// TIA Portal project "FactoryIO_Template_S7-1500_V15" (V15)

(* hardware
DEVICE "S71500/ET200MP-Station_1"  S7-1500 station
   slot 0: "Profilschiene_0"  6ES7 590-1***0-0AA0
   slot 1: "PLC_1"  CPU 1511-1 PN  6ES7 511-1AK00-0AB0  V1.8
   slot 2: "AI 8xU/I/RTD/TC ST_1"  AI 8xU/I/RTD/TC ST  6ES7 531-7KF00-0AB0  V2.0
   slot 3: "AI 8xU/I/RTD/TC ST_2"  AI 8xU/I/RTD/TC ST  6ES7 531-7KF00-0AB0  V2.0
   slot 4: "AI 8xU/I/RTD/TC ST_3"  AI 8xU/I/RTD/TC ST  6ES7 531-7KF00-0AB0  V2.0
   slot 5: "AI 8xU/I/RTD/TC ST_4"  AI 8xU/I/RTD/TC ST  6ES7 531-7KF00-0AB0  V2.0
   slot 6: "DI 16x24VDC BA_1"  DI 16x24VDC BA  6ES7 521-1BH10-0AA0  V1.0
*)

// ===== PLC "PLC_1"  CPU 1511-1 PN =====

VAR_GLOBAL   // PLC tag table "Standard-Variablentabelle"
   "counter green" AT %QD31 : UDInt;
END_VAR

VAR_GLOBAL   // PLC tag table "Input tag table"
   "start" AT %I0.0 : Bool;
   "stop" AT %I0.1 : Bool;
   "reset" AT %I0.2 : Bool;
   "emergency" AT %I0.3 : Bool;
   "right 1 limit" AT %I0.4 : Bool;
   "right 1 clamped" AT %I0.5 : Bool;
   "right 2 limit" AT %I0.6 : Bool;
   "right 2 clamped" AT %I0.7 : Bool;
   "mc1 opened" AT %I1.0 : Bool;
   "mc1 busy" AT %I1.1 : Bool;
   "mc1 error" AT %I1.2 : Bool;
   "mc2 opened" AT %I1.3 : Bool;
   "mc2 busy" AT %I1.4 : Bool;
   "mc2 error" AT %I1.5 : Bool;
   "mc3 opened" AT %I1.6 : Bool;
   "mc3 busy" AT %I1.7 : Bool;
   "mc3 error" AT %I2.0 : Bool;
   "mc5 opened" AT %I2.1 : Bool;
   "mc5 busy" AT %I2.2 : Bool;
   "mc5 error" AT %I2.3 : Bool;
   "pusher 3 front limit" AT %I2.4 : Bool;
   "pusher 1 front limit" AT %I2.5 : Bool;
   "pusher 4 front limit" AT %I2.6 : Bool;
   "pusher 2 front limit" AT %I2.7 : Bool;
   "right 3 limit" AT %I3.0 : Bool;
   "right 3 clamped" AT %I3.1 : Bool;
   "right 5 limit" AT %I3.2 : Bool;
   "right 5 clamped" AT %I3.3 : Bool;
   "axis 1 detected" AT %I3.4 : Bool;
   "axis 1 moving z" AT %I3.5 : Bool;
   "axis 1 moving x" AT %I3.6 : Bool;
   "axis 2 detected" AT %I3.7 : Bool;
   "axis 2 moving z" AT %I4.0 : Bool;
   "axis 2 moving x" AT %I4.1 : Bool;
   "vision sensor 1" AT %I4.2 : Bool;
   "vision sensor 2" AT %I4.3 : Bool;
   "vision sensor 3" AT %I4.4 : Bool;
   "vision sensor 4" AT %I4.5 : Bool;
   "diffuser sensor 1" AT %I4.6 : Bool;
   "diffuser sensor 2" AT %I4.7 : Bool;
   "diffuser sensor 3" AT %I5.0 : Bool;
   "diffuser sensor 4" AT %I5.1 : Bool;
   "diffuser sensor 5" AT %I5.2 : Bool;
   "diffuser sensor 6" AT %I5.3 : Bool;
END_VAR

VAR_GLOBAL   // PLC tag table "Memory tag table"
   "start memory" AT %M0.0 : Bool;
   "stop memory" AT %M0.1 : Bool;
   "Tag_1" AT %M0.2 : Bool;
   "Tag_2" AT %M0.3 : Bool;
   "Tag_3" AT %M0.4 : Bool;
   "Tag_4" AT %M0.5 : Bool;
   "Tag_5" AT %M0.6 : Bool;
   "Tag_6" AT %M0.7 : Bool;
   "Lid alined" AT %M1.0 : Bool;
   "Tag_7" AT %M1.1 : Bool;
   "Tag_8" AT %M1.2 : Bool;
   "base alined" AT %M1.3 : Bool;
   "Tag_9" AT %M1.4 : Bool;
   "MOVE Z BIT" AT %M1.5 : Bool;
   "Tag_10" AT %M1.6 : Bool;
   "Tag_11" AT %M1.7 : Bool;
   "Tag_12" AT %M2.0 : Bool;
   "Tag_13" AT %M2.1 : Bool;
   "Tag_14" AT %M2.2 : Bool;
   "MOVE Z BIT 2" AT %M2.3 : Bool;
   "Tag_15" AT %M2.4 : Bool;
   "TEMPORARY" AT %M2.5 : Bool;
   "Tag_16" AT %M2.6 : Bool;
   "TEMPORARY 2" AT %M2.7 : Bool;
   "Tag_17" AT %M3.0 : Bool;
   "Tag_1(1)" AT %M3.1 : Bool;
   "Tag_2(1)" AT %M3.2 : Bool;
   "Tag_3(1)" AT %M3.3 : Bool;
   "Tag_4(1)" AT %M3.4 : Bool;
   "Tag_5(1)" AT %M3.5 : Bool;
   "Tag_6(1)" AT %M3.6 : Bool;
   "Lid alined(1)" AT %M3.7 : Bool;
   "Tag_7(1)" AT %M4.0 : Bool;
   "Tag_8(1)" AT %M4.1 : Bool;
   "base alined(1)" AT %M4.2 : Bool;
   "Tag_9(1)" AT %M4.3 : Bool;
   "MOVE Z BIT(1)" AT %M4.4 : Bool;
   "Tag_10(1)" AT %M4.5 : Bool;
   "Tag_11(1)" AT %M4.6 : Bool;
   "Tag_12(1)" AT %M4.7 : Bool;
   "Tag_13(1)" AT %M5.0 : Bool;
   "Tag_14(1)" AT %M5.1 : Bool;
   "MOVE Z BIT 2(1)" AT %M5.2 : Bool;
   "Tag_15(1)" AT %M5.3 : Bool;
   "TEMPORARY(1)" AT %M5.4 : Bool;
   "Tag_16(1)" AT %M5.5 : Bool;
   "TEMPORARY 2(1)" AT %M5.6 : Bool;
   "Tag_17(1)" AT %M5.7 : Bool;
   "tag 18" AT %M6.0 : Bool;
END_VAR

VAR_GLOBAL   // PLC tag table "Output tag table"
   "belt conveyor (2m)1" AT %Q0.0 : Bool;
   "belt conveyor (2m)2" AT %Q0.1 : Bool;
   "belt conveyor (2m)3" AT %Q0.2 : Bool;
   "belt conveyor (2m)5" AT %Q0.3 : Bool;
   "belt conveyor (2m)7" AT %Q0.4 : Bool;
   "belt conveyor (2m)9" AT %Q0.5 : Bool;
   "belt conveyor (2m)14" AT %Q0.6 : Bool;
   "belt conveyor (4m)2" AT %Q1.0 : Bool;
   "belt conveyor (4m)4" AT %Q1.1 : Bool;
   "belt conveyor (6m)1" AT %Q1.2 : Bool;
   "emitter 2" AT %Q1.3 : Bool;
   "emitter 3" AT %Q1.4 : Bool;
   "emitter 4" AT %Q1.5 : Bool;
   "emitter 6" AT %Q1.6 : Bool;
   "factory pause" AT %Q1.7 : Bool;
   "factory reset" AT %Q2.0 : Bool;
   "right 1 clamp" AT %Q2.1 : Bool;
   "right 1 raise" AT %Q2.2 : Bool;
   "right 2 clamp" AT %Q2.3 : Bool;
   "right 2 raise" AT %Q2.4 : Bool;
   "mc1 start" AT %Q2.5 : Bool;
   "mc1 stop" AT %Q2.6 : Bool;
   "mc1 reset" AT %Q2.7 : Bool;
   "mc1 producing leds" AT %Q3.0 : Bool;
   "mc2 start" AT %Q3.1 : Bool;
   "mc2 stop" AT %Q3.2 : Bool;
   "mc2 reset" AT %Q3.3 : Bool;
   "mc2 producing leds" AT %Q3.4 : Bool;
   "mc3 start" AT %Q3.5 : Bool;
   "mc3 stop" AT %Q3.6 : Bool;
   "mc3 reset" AT %Q3.7 : Bool;
   "mc3 producing leds" AT %Q4.0 : Bool;
   "mc5 start" AT %Q4.1 : Bool;
   "mc5 stop" AT %Q4.2 : Bool;
   "mc5 reset" AT %Q4.3 : Bool;
   "mc5 producing leds" AT %Q4.4 : Bool;
   "pusher 1" AT %Q4.5 : Bool;
   "pusher 2" AT %Q4.6 : Bool;
   "remover 1" AT %Q4.7 : Bool;
   "remover 2" AT %Q5.0 : Bool;
   "reset light" AT %Q5.1 : Bool;
   "start light" AT %Q5.2 : Bool;
   "stop light" AT %Q5.3 : Bool;
   "right 3 clamp" AT %Q5.4 : Bool;
   "right 3 raise" AT %Q5.5 : Bool;
   "right 5 clamp" AT %Q5.6 : Bool;
   "right 5 raise" AT %Q5.7 : Bool;
   "axis 1 x" AT %Q6.0 : Bool;
   "axis 1 z" AT %Q6.1 : Bool;
   "axis 1 grab" AT %Q6.2 : Bool;
   "axis 2 x" AT %Q6.3 : Bool;
   "axis 2 z" AT %Q6.4 : Bool;
   "axis 2 grab" AT %Q6.5 : Bool;
   "belt conveyor (4m)1" AT %Q6.6 : Bool;
   "belt conveyor (6m)2" AT %Q6.7 : Bool;
   "belt conveyor (6m)3" AT %Q7.0 : Bool;
   "belt conveyor (6m)4" AT %Q7.1 : Bool;
   "belt conveyor (6m)5" AT %Q7.2 : Bool;
   "belt conveyor (6m)6" AT %Q7.3 : Bool;
   "pusher 3" AT %Q7.4 : Bool;
   "pusher 4" AT %Q7.5 : Bool;
   "counter blue" AT %QD8 : UDInt;
   "counter 2" AT %QD12 : UDInt;
END_VAR

// folder: System blocks/Program resources

DATA_BLOCK "IEC_Timer_0_DB"   // DB1
{ S7_Optimized_Access := 'TRUE' }
AUTHOR : Simatic
FAMILY : IEC
NAME : IEC_TMR
VERSION : 1.0
// stored: InstanceOfName IEC_TIMER
"IEC_TIMER"
BEGIN
END_DATA_BLOCK

DATA_BLOCK "IEC_Timer_0_DB_1"   // DB2
{ S7_Optimized_Access := 'TRUE' }
AUTHOR : Simatic
FAMILY : IEC
NAME : IEC_TMR
VERSION : 1.0
// stored: InstanceOfName IEC_TIMER
"IEC_TIMER"
BEGIN
END_DATA_BLOCK

DATA_BLOCK "IEC_Timer_0_DB_2"   // DB3
{ S7_Optimized_Access := 'TRUE' }
AUTHOR : Simatic
FAMILY : IEC
NAME : IEC_TMR
VERSION : 1.0
// stored: InstanceOfName IEC_TIMER
"IEC_TIMER"
BEGIN
END_DATA_BLOCK

DATA_BLOCK "IEC_Timer_0_DB_3"   // DB4
{ S7_Optimized_Access := 'TRUE' }
AUTHOR : Simatic
FAMILY : IEC
NAME : IEC_TMR
VERSION : 1.0
// stored: InstanceOfName IEC_TIMER
"IEC_TIMER"
BEGIN
END_DATA_BLOCK

DATA_BLOCK "IEC_Timer_0_DB_4"   // DB5
{ S7_Optimized_Access := 'TRUE' }
AUTHOR : Simatic
FAMILY : IEC
NAME : IEC_TMR
VERSION : 1.0
// stored: InstanceOfName IEC_TIMER
"IEC_TIMER"
BEGIN
END_DATA_BLOCK

DATA_BLOCK "IEC_Timer_0_DB_6"   // DB6
{ S7_Optimized_Access := 'TRUE' }
AUTHOR : Simatic
FAMILY : IEC
NAME : IEC_TMR
VERSION : 1.0
// stored: InstanceOfName IEC_TIMER
"IEC_TIMER"
BEGIN
END_DATA_BLOCK

// folder: (top level)

FUNCTION "blue belt conveyor" : Void   // FC1, LAD
{ S7_Optimized_Access := 'TRUE' }
VERSION : 0.1
   VAR_TEMP   // added for the SCL form of the ladder/FBD networks
      _w1 : Bool;
   END_VAR
BEGIN

REGION Network 1
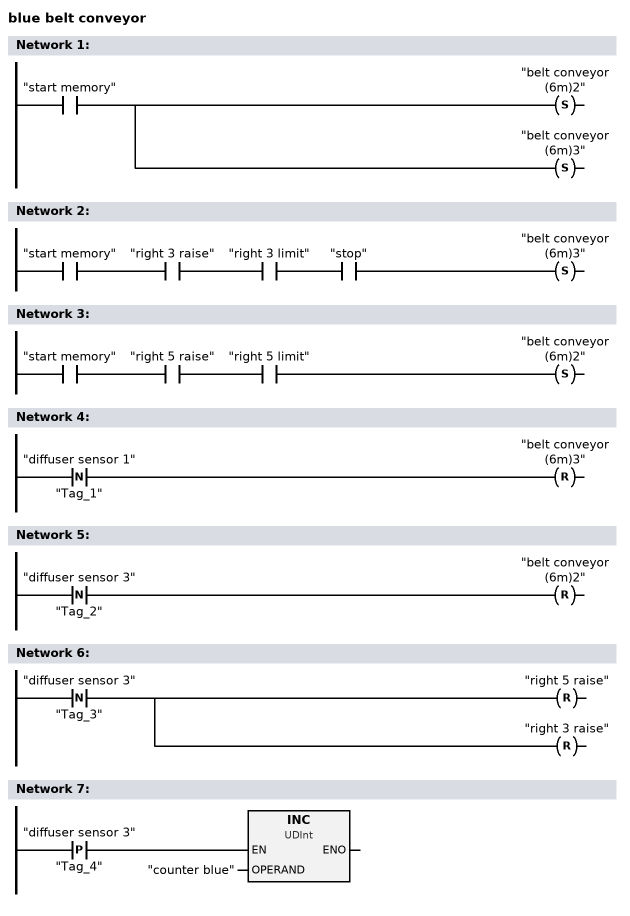
   RUNG wire#powerrail
      Contact( "start memory" )
      wire#w1
      S_Coil( "belt conveyor (6m)2" )
   END_RUNG
   RUNG wire#w1
      S_Coil( "belt conveyor (6m)3" )
   END_RUNG
   // the same network as SCL:
   IF "start memory" THEN
       "belt conveyor (6m)2" := TRUE;
       "belt conveyor (6m)3" := TRUE;
   END_IF;
END_REGION

REGION Network 2
   RUNG wire#powerrail
      Contact( "start memory" )
      Contact( "right 3 raise" )
      Contact( "right 3 limit" )
      Contact( "stop" )
      S_Coil( "belt conveyor (6m)3" )
   END_RUNG
   // the same network as SCL:
   IF "start memory" AND "right 3 raise" AND "right 3 limit" AND "stop" THEN
       "belt conveyor (6m)3" := TRUE;
   END_IF;
END_REGION

REGION Network 3
   RUNG wire#powerrail
      Contact( "start memory" )
      Contact( "right 5 raise" )
      Contact( "right 5 limit" )
      S_Coil( "belt conveyor (6m)2" )
   END_RUNG
   // the same network as SCL:
   IF "start memory" AND "right 5 raise" AND "right 5 limit" THEN "belt conveyor (6m)2" := TRUE; END_IF;
END_REGION

REGION Network 4
   RUNG wire#powerrail
      N_Contact(operand := "diffuser sensor 1", bit := "Tag_1")
      R_Coil( "belt conveyor (6m)3" )
   END_RUNG
   // the same network as SCL:
   #_w1 := NOT "diffuser sensor 1" AND "Tag_1";   // falling edge of "diffuser sensor 1"
   "Tag_1" := "diffuser sensor 1";
   IF #_w1 THEN "belt conveyor (6m)3" := FALSE; END_IF;
END_REGION

REGION Network 5
   RUNG wire#powerrail
      N_Contact(operand := "diffuser sensor 3", bit := "Tag_2")
      R_Coil( "belt conveyor (6m)2" )
   END_RUNG
   // the same network as SCL:
   #_w1 := NOT "diffuser sensor 3" AND "Tag_2";   // falling edge of "diffuser sensor 3"
   "Tag_2" := "diffuser sensor 3";
   IF #_w1 THEN "belt conveyor (6m)2" := FALSE; END_IF;
END_REGION

REGION Network 6
   RUNG wire#powerrail
      N_Contact(operand := "diffuser sensor 3", bit := "Tag_3")
      wire#w1
      R_Coil( "right 5 raise" )
   END_RUNG
   RUNG wire#w1
      R_Coil( "right 3 raise" )
   END_RUNG
   // the same network as SCL:
   #_w1 := NOT "diffuser sensor 3" AND "Tag_3";   // falling edge of "diffuser sensor 3"
   "Tag_3" := "diffuser sensor 3";
   IF #_w1 THEN
       "right 5 raise" := FALSE;
       "right 3 raise" := FALSE;
   END_IF;
END_REGION

REGION Network 7
   RUNG wire#powerrail
      P_Contact(operand := "diffuser sensor 3", bit := "Tag_4")
      { S7_Templates := "DestType := UDInt" } Inc( "counter blue" )
   END_RUNG
   // the same network as SCL:
   #_w1 := "diffuser sensor 3" AND NOT "Tag_4";   // rising edge of "diffuser sensor 3"
   "Tag_4" := "diffuser sensor 3";
   IF #_w1 THEN "counter blue" := "counter blue" + 1; END_IF;
END_REGION
END_FUNCTION

FUNCTION "blue Clamp" : Void   // FC2, LAD
{ S7_Optimized_Access := 'TRUE' }
VERSION : 0.1
   VAR_TEMP   // added for the SCL form of the ladder/FBD networks
      _w1 : Bool;
   END_VAR
BEGIN

REGION Network 1
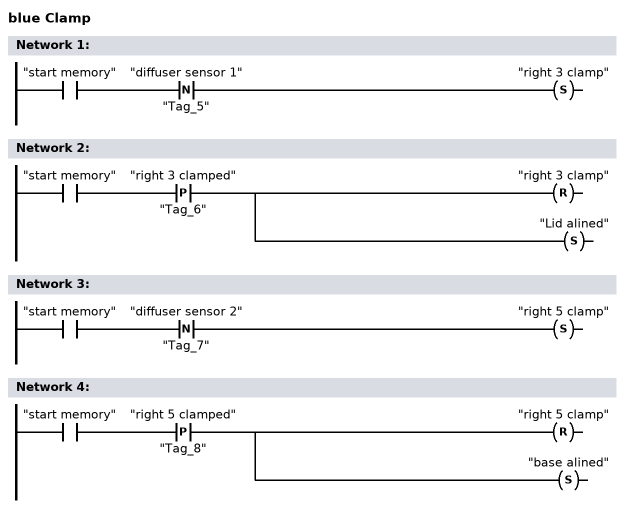
   RUNG wire#powerrail
      Contact( "start memory" )
      N_Contact(operand := "diffuser sensor 1", bit := "Tag_5")
      S_Coil( "right 3 clamp" )
   END_RUNG
   // the same network as SCL:
   #_w1 := "start memory" AND NOT "diffuser sensor 1" AND "Tag_5";   // falling edge of "diffuser sensor 1"
   "Tag_5" := "diffuser sensor 1";
   IF #_w1 THEN "right 3 clamp" := TRUE; END_IF;
END_REGION

REGION Network 2
   RUNG wire#powerrail
      Contact( "start memory" )
      P_Contact(operand := "right 3 clamped", bit := "Tag_6")
      wire#w1
      R_Coil( "right 3 clamp" )
   END_RUNG
   RUNG wire#w1
      S_Coil( "Lid alined" )
   END_RUNG
   // the same network as SCL:
   #_w1 := "start memory" AND "right 3 clamped" AND NOT "Tag_6";   // rising edge of "right 3 clamped"
   "Tag_6" := "right 3 clamped";
   IF #_w1 THEN
       "right 3 clamp" := FALSE;
       "Lid alined" := TRUE;
   END_IF;
END_REGION

REGION Network 3
   RUNG wire#powerrail
      Contact( "start memory" )
      N_Contact(operand := "diffuser sensor 2", bit := "Tag_7")
      S_Coil( "right 5 clamp" )
   END_RUNG
   // the same network as SCL:
   #_w1 := "start memory" AND NOT "diffuser sensor 2" AND "Tag_7";   // falling edge of "diffuser sensor 2"
   "Tag_7" := "diffuser sensor 2";
   IF #_w1 THEN "right 5 clamp" := TRUE; END_IF;
END_REGION

REGION Network 4
   RUNG wire#powerrail
      Contact( "start memory" )
      P_Contact(operand := "right 5 clamped", bit := "Tag_8")
      wire#w1
      R_Coil( "right 5 clamp" )
   END_RUNG
   RUNG wire#w1
      S_Coil( "base alined" )
   END_RUNG
   // the same network as SCL:
   #_w1 := "start memory" AND "right 5 clamped" AND NOT "Tag_8";   // rising edge of "right 5 clamped"
   "Tag_8" := "right 5 clamped";
   IF #_w1 THEN
       "right 5 clamp" := FALSE;
       "base alined" := TRUE;
   END_IF;
END_REGION
END_FUNCTION

FUNCTION "blue pICK & pLACE" : Void   // FC3, LAD
{ S7_Optimized_Access := 'TRUE' }
VERSION : 0.1
   VAR_TEMP   // added for the SCL form of the ladder/FBD networks
      _w1 : Bool;
   END_VAR
BEGIN

REGION Network 1
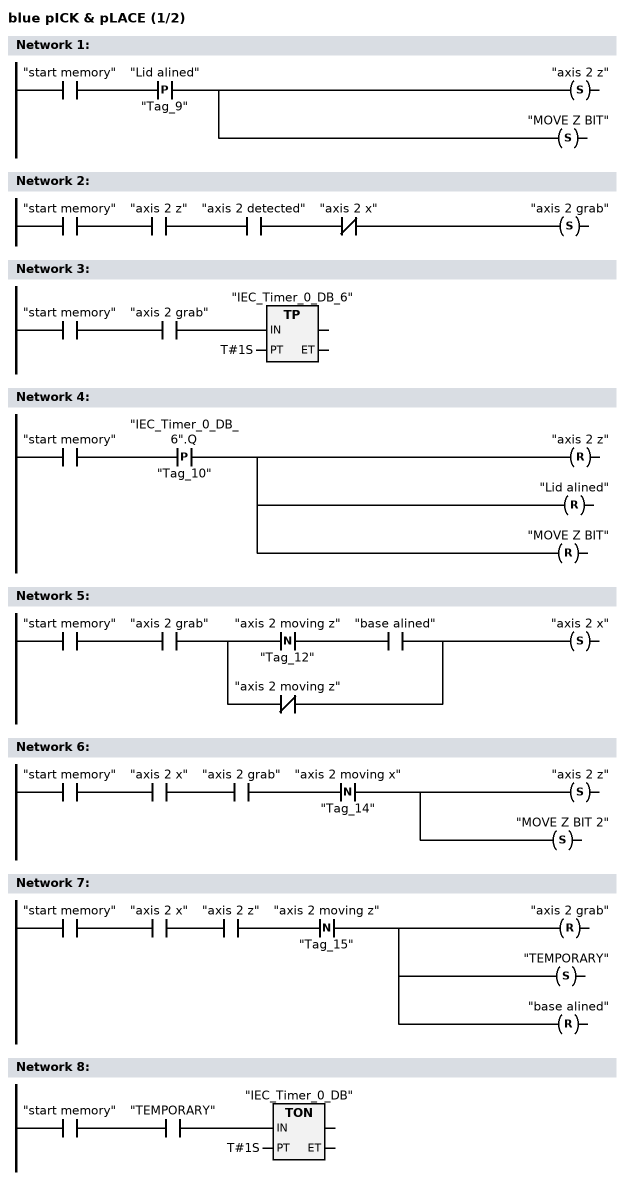
   RUNG wire#powerrail
      Contact( "start memory" )
      P_Contact(operand := "Lid alined", bit := "Tag_9")
      wire#w1
      S_Coil( "axis 2 z" )
   END_RUNG
   RUNG wire#w1
      S_Coil( "MOVE Z BIT" )
   END_RUNG
   // the same network as SCL:
   #_w1 := "start memory" AND "Lid alined" AND NOT "Tag_9";   // rising edge of "Lid alined"
   "Tag_9" := "Lid alined";
   IF #_w1 THEN
       "axis 2 z" := TRUE;
       "MOVE Z BIT" := TRUE;
   END_IF;
END_REGION

REGION Network 2
   RUNG wire#powerrail
      Contact( "start memory" )
      Contact( "axis 2 z" )
      Contact( "axis 2 detected" )
      I_Contact( "axis 2 x" )
      S_Coil( "axis 2 grab" )
   END_RUNG
   // the same network as SCL:
   IF "start memory" AND "axis 2 z" AND "axis 2 detected" AND NOT "axis 2 x" THEN
       "axis 2 grab" := TRUE;
   END_IF;
END_REGION

REGION Network 3
   "IEC_Timer_0_DB_6".TP(IN := "start memory" AND "axis 2 grab", PT := T#1S);
END_REGION

REGION Network 4
   RUNG wire#powerrail
      Contact( "start memory" )
      P_Contact(operand := "IEC_Timer_0_DB_6".Q, bit := "Tag_10")
      wire#w1
      R_Coil( "axis 2 z" )
   END_RUNG
   RUNG wire#w1
      R_Coil( "Lid alined" )
   END_RUNG
   RUNG wire#w1
      R_Coil( "MOVE Z BIT" )
   END_RUNG
   // the same network as SCL:
   #_w1 := "start memory" AND "IEC_Timer_0_DB_6".Q AND NOT "Tag_10";   // rising edge of "IEC_Timer_0_DB_6".Q
   "Tag_10" := "IEC_Timer_0_DB_6".Q;
   IF #_w1 THEN
       "axis 2 z" := FALSE;
       "Lid alined" := FALSE;
       "MOVE Z BIT" := FALSE;
   END_IF;
END_REGION

REGION Network 5
   RUNG wire#powerrail
      Contact( "start memory" )
      Contact( "axis 2 grab" )
      wire#w1
      N_Contact(operand := "axis 2 moving z", bit := "Tag_12")
      Contact( "base alined" )
      wire#w2
      S_Coil( "axis 2 x" )
   END_RUNG
   RUNG wire#w1
      I_Contact( "axis 2 moving z" )
   END_RUNG wire#w2
   // the same network as SCL:
   #_w1 := "start memory" AND "axis 2 grab" AND NOT "axis 2 moving z" AND "Tag_12";   // falling edge of "axis 2 moving z"
   "Tag_12" := "axis 2 moving z";
   IF (#_w1 AND "base alined") OR ("start memory" AND "axis 2 grab" AND NOT "axis 2 moving z") THEN
       "axis 2 x" := TRUE;
   END_IF;
END_REGION

REGION Network 6
   RUNG wire#powerrail
      Contact( "start memory" )
      Contact( "axis 2 x" )
      Contact( "axis 2 grab" )
      N_Contact(operand := "axis 2 moving x", bit := "Tag_14")
      wire#w1
      S_Coil( "axis 2 z" )
   END_RUNG
   RUNG wire#w1
      S_Coil( "MOVE Z BIT 2" )
   END_RUNG
   // the same network as SCL:
   #_w1 := "start memory" AND "axis 2 x" AND "axis 2 grab" AND NOT "axis 2 moving x" AND "Tag_14";   // falling edge of "axis 2 moving x"
   "Tag_14" := "axis 2 moving x";
   IF #_w1 THEN
       "axis 2 z" := TRUE;
       "MOVE Z BIT 2" := TRUE;
   END_IF;
END_REGION

REGION Network 7
   RUNG wire#powerrail
      Contact( "start memory" )
      Contact( "axis 2 x" )
      Contact( "axis 2 z" )
      N_Contact(operand := "axis 2 moving z", bit := "Tag_15")
      wire#w1
      R_Coil( "axis 2 grab" )
   END_RUNG
   RUNG wire#w1
      S_Coil( "TEMPORARY" )
   END_RUNG
   RUNG wire#w1
      R_Coil( "base alined" )
   END_RUNG
   // the same network as SCL:
   #_w1 := "start memory" AND "axis 2 x" AND "axis 2 z" AND NOT "axis 2 moving z" AND "Tag_15";   // falling edge of "axis 2 moving z"
   "Tag_15" := "axis 2 moving z";
   IF #_w1 THEN
       "axis 2 grab" := FALSE;
       "TEMPORARY" := TRUE;
       "base alined" := FALSE;
   END_IF;
END_REGION

REGION Network 8
   "IEC_Timer_0_DB".TON(IN := "start memory" AND "TEMPORARY", PT := T#1S);
END_REGION

REGION Network 9
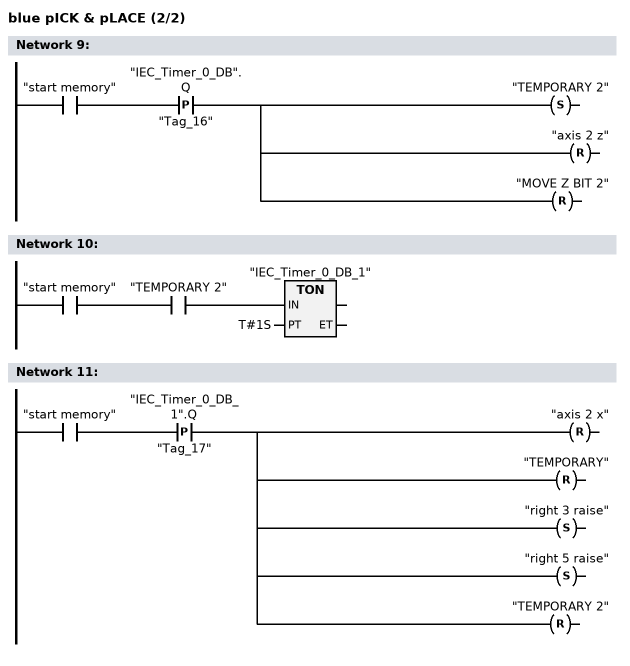
   RUNG wire#powerrail
      Contact( "start memory" )
      P_Contact(operand := "IEC_Timer_0_DB".Q, bit := "Tag_16")
      wire#w1
      S_Coil( "TEMPORARY 2" )
   END_RUNG
   RUNG wire#w1
      R_Coil( "axis 2 z" )
   END_RUNG
   RUNG wire#w1
      R_Coil( "MOVE Z BIT 2" )
   END_RUNG
   // the same network as SCL:
   #_w1 := "start memory" AND "IEC_Timer_0_DB".Q AND NOT "Tag_16";   // rising edge of "IEC_Timer_0_DB".Q
   "Tag_16" := "IEC_Timer_0_DB".Q;
   IF #_w1 THEN
       "TEMPORARY 2" := TRUE;
       "axis 2 z" := FALSE;
       "MOVE Z BIT 2" := FALSE;
   END_IF;
END_REGION

REGION Network 10
   "IEC_Timer_0_DB_1".TON(IN := "start memory" AND "TEMPORARY 2", PT := T#1S);
END_REGION

REGION Network 11
   RUNG wire#powerrail
      Contact( "start memory" )
      P_Contact(operand := "IEC_Timer_0_DB_1".Q, bit := "Tag_17")
      wire#w1
      R_Coil( "axis 2 x" )
   END_RUNG
   RUNG wire#w1
      R_Coil( "TEMPORARY" )
   END_RUNG
   RUNG wire#w1
      S_Coil( "right 3 raise" )
   END_RUNG
   RUNG wire#w1
      S_Coil( "right 5 raise" )
   END_RUNG
   RUNG wire#w1
      R_Coil( "TEMPORARY 2" )
   END_RUNG
   // the same network as SCL:
   #_w1 := "start memory" AND "IEC_Timer_0_DB_1".Q AND NOT "Tag_17";   // rising edge of "IEC_Timer_0_DB_1".Q
   "Tag_17" := "IEC_Timer_0_DB_1".Q;
   IF #_w1 THEN
       "axis 2 x" := FALSE;
       "TEMPORARY" := FALSE;
       "right 3 raise" := TRUE;
       "right 5 raise" := TRUE;
       "TEMPORARY 2" := FALSE;
   END_IF;
END_REGION
END_FUNCTION

FUNCTION "green belt conveyor" : Void   // FC4, LAD
{ S7_Optimized_Access := 'TRUE' }
VERSION : 0.1
   VAR_TEMP   // added for the SCL form of the ladder/FBD networks
      _w1 : Bool;
   END_VAR
BEGIN

REGION Network 1
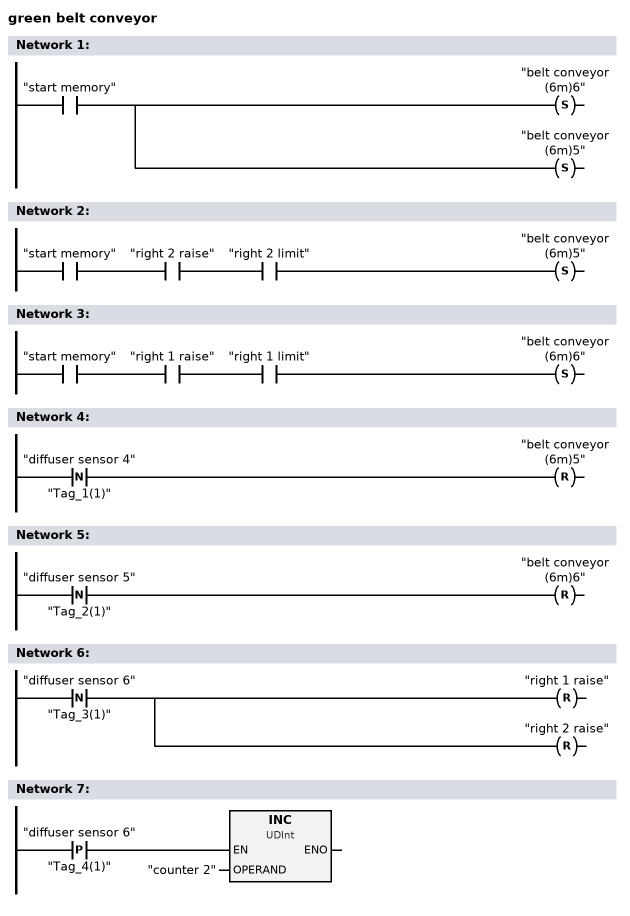
   RUNG wire#powerrail
      Contact( "start memory" )
      wire#w1
      S_Coil( "belt conveyor (6m)6" )
   END_RUNG
   RUNG wire#w1
      S_Coil( "belt conveyor (6m)5" )
   END_RUNG
   // the same network as SCL:
   IF "start memory" THEN
       "belt conveyor (6m)6" := TRUE;
       "belt conveyor (6m)5" := TRUE;
   END_IF;
END_REGION

REGION Network 2
   RUNG wire#powerrail
      Contact( "start memory" )
      Contact( "right 2 raise" )
      Contact( "right 2 limit" )
      S_Coil( "belt conveyor (6m)5" )
   END_RUNG
   // the same network as SCL:
   IF "start memory" AND "right 2 raise" AND "right 2 limit" THEN "belt conveyor (6m)5" := TRUE; END_IF;
END_REGION

REGION Network 3
   RUNG wire#powerrail
      Contact( "start memory" )
      Contact( "right 1 raise" )
      Contact( "right 1 limit" )
      S_Coil( "belt conveyor (6m)6" )
   END_RUNG
   // the same network as SCL:
   IF "start memory" AND "right 1 raise" AND "right 1 limit" THEN "belt conveyor (6m)6" := TRUE; END_IF;
END_REGION

REGION Network 4
   RUNG wire#powerrail
      N_Contact(operand := "diffuser sensor 4", bit := "Tag_1(1)")
      R_Coil( "belt conveyor (6m)5" )
   END_RUNG
   // the same network as SCL:
   #_w1 := NOT "diffuser sensor 4" AND "Tag_1(1)";   // falling edge of "diffuser sensor 4"
   "Tag_1(1)" := "diffuser sensor 4";
   IF #_w1 THEN "belt conveyor (6m)5" := FALSE; END_IF;
END_REGION

REGION Network 5
   RUNG wire#powerrail
      N_Contact(operand := "diffuser sensor 5", bit := "Tag_2(1)")
      R_Coil( "belt conveyor (6m)6" )
   END_RUNG
   // the same network as SCL:
   #_w1 := NOT "diffuser sensor 5" AND "Tag_2(1)";   // falling edge of "diffuser sensor 5"
   "Tag_2(1)" := "diffuser sensor 5";
   IF #_w1 THEN "belt conveyor (6m)6" := FALSE; END_IF;
END_REGION

REGION Network 6
   RUNG wire#powerrail
      N_Contact(operand := "diffuser sensor 6", bit := "Tag_3(1)")
      wire#w1
      R_Coil( "right 1 raise" )
   END_RUNG
   RUNG wire#w1
      R_Coil( "right 2 raise" )
   END_RUNG
   // the same network as SCL:
   #_w1 := NOT "diffuser sensor 6" AND "Tag_3(1)";   // falling edge of "diffuser sensor 6"
   "Tag_3(1)" := "diffuser sensor 6";
   IF #_w1 THEN
       "right 1 raise" := FALSE;
       "right 2 raise" := FALSE;
   END_IF;
END_REGION

REGION Network 7
   RUNG wire#powerrail
      P_Contact(operand := "diffuser sensor 6", bit := "Tag_4(1)")
      { S7_Templates := "DestType := UDInt" } Inc( "counter 2" )
   END_RUNG
   // the same network as SCL:
   #_w1 := "diffuser sensor 6" AND NOT "Tag_4(1)";   // rising edge of "diffuser sensor 6"
   "Tag_4(1)" := "diffuser sensor 6";
   IF #_w1 THEN "counter 2" := "counter 2" + 1; END_IF;
END_REGION
END_FUNCTION

FUNCTION "green Clamp" : Void   // FC5, LAD
{ S7_Optimized_Access := 'TRUE' }
VERSION : 0.1
   VAR_TEMP   // added for the SCL form of the ladder/FBD networks
      _w1 : Bool;
   END_VAR
BEGIN

REGION Network 1
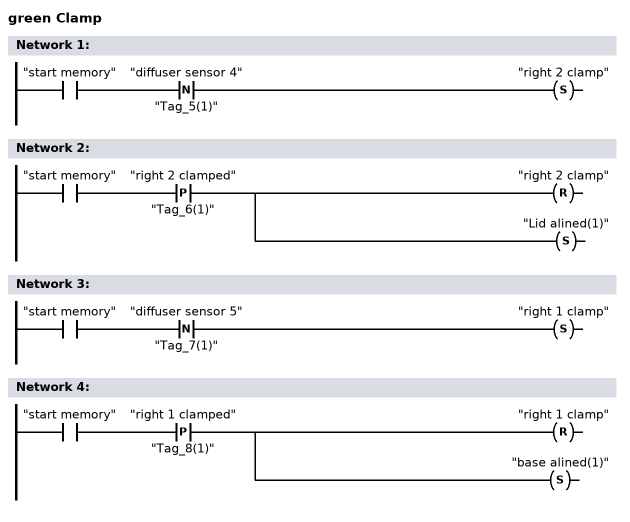
   RUNG wire#powerrail
      Contact( "start memory" )
      N_Contact(operand := "diffuser sensor 4", bit := "Tag_5(1)")
      S_Coil( "right 2 clamp" )
   END_RUNG
   // the same network as SCL:
   #_w1 := "start memory" AND NOT "diffuser sensor 4" AND "Tag_5(1)";   // falling edge of "diffuser sensor 4"
   "Tag_5(1)" := "diffuser sensor 4";
   IF #_w1 THEN "right 2 clamp" := TRUE; END_IF;
END_REGION

REGION Network 2
   RUNG wire#powerrail
      Contact( "start memory" )
      P_Contact(operand := "right 2 clamped", bit := "Tag_6(1)")
      wire#w1
      R_Coil( "right 2 clamp" )
   END_RUNG
   RUNG wire#w1
      S_Coil( "Lid alined(1)" )
   END_RUNG
   // the same network as SCL:
   #_w1 := "start memory" AND "right 2 clamped" AND NOT "Tag_6(1)";   // rising edge of "right 2 clamped"
   "Tag_6(1)" := "right 2 clamped";
   IF #_w1 THEN
       "right 2 clamp" := FALSE;
       "Lid alined(1)" := TRUE;
   END_IF;
END_REGION

REGION Network 3
   RUNG wire#powerrail
      Contact( "start memory" )
      N_Contact(operand := "diffuser sensor 5", bit := "Tag_7(1)")
      S_Coil( "right 1 clamp" )
   END_RUNG
   // the same network as SCL:
   #_w1 := "start memory" AND NOT "diffuser sensor 5" AND "Tag_7(1)";   // falling edge of "diffuser sensor 5"
   "Tag_7(1)" := "diffuser sensor 5";
   IF #_w1 THEN "right 1 clamp" := TRUE; END_IF;
END_REGION

REGION Network 4
   RUNG wire#powerrail
      Contact( "start memory" )
      P_Contact(operand := "right 1 clamped", bit := "Tag_8(1)")
      wire#w1
      R_Coil( "right 1 clamp" )
   END_RUNG
   RUNG wire#w1
      S_Coil( "base alined(1)" )
   END_RUNG
   // the same network as SCL:
   #_w1 := "start memory" AND "right 1 clamped" AND NOT "Tag_8(1)";   // rising edge of "right 1 clamped"
   "Tag_8(1)" := "right 1 clamped";
   IF #_w1 THEN
       "right 1 clamp" := FALSE;
       "base alined(1)" := TRUE;
   END_IF;
END_REGION
END_FUNCTION

FUNCTION "green pICK & pLACE" : Void   // FC6, LAD
{ S7_Optimized_Access := 'TRUE' }
VERSION : 0.1
   VAR_TEMP   // added for the SCL form of the ladder/FBD networks
      _w1 : Bool;
   END_VAR
BEGIN

REGION Network 1
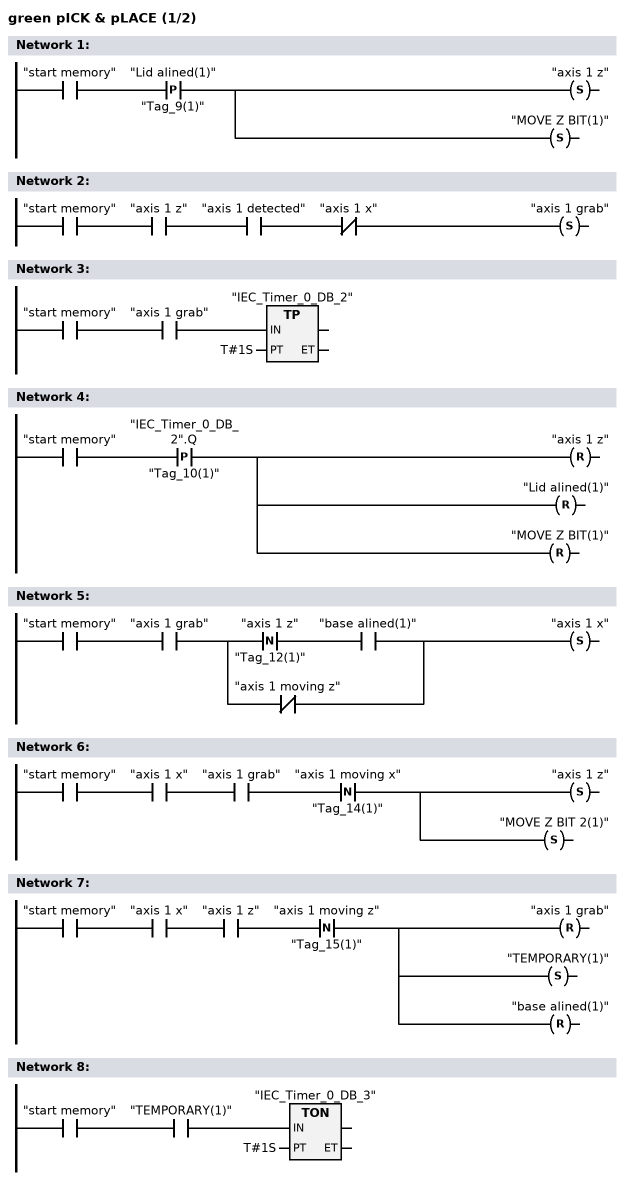
   RUNG wire#powerrail
      Contact( "start memory" )
      P_Contact(operand := "Lid alined(1)", bit := "Tag_9(1)")
      wire#w1
      S_Coil( "axis 1 z" )
   END_RUNG
   RUNG wire#w1
      S_Coil( "MOVE Z BIT(1)" )
   END_RUNG
   // the same network as SCL:
   #_w1 := "start memory" AND "Lid alined(1)" AND NOT "Tag_9(1)";   // rising edge of "Lid alined(1)"
   "Tag_9(1)" := "Lid alined(1)";
   IF #_w1 THEN
       "axis 1 z" := TRUE;
       "MOVE Z BIT(1)" := TRUE;
   END_IF;
END_REGION

REGION Network 2
   RUNG wire#powerrail
      Contact( "start memory" )
      Contact( "axis 1 z" )
      Contact( "axis 1 detected" )
      I_Contact( "axis 1 x" )
      S_Coil( "axis 1 grab" )
   END_RUNG
   // the same network as SCL:
   IF "start memory" AND "axis 1 z" AND "axis 1 detected" AND NOT "axis 1 x" THEN
       "axis 1 grab" := TRUE;
   END_IF;
END_REGION

REGION Network 3
   "IEC_Timer_0_DB_2".TP(IN := "start memory" AND "axis 1 grab", PT := T#1S);
END_REGION

REGION Network 4
   RUNG wire#powerrail
      Contact( "start memory" )
      P_Contact(operand := "IEC_Timer_0_DB_2".Q, bit := "Tag_10(1)")
      wire#w1
      R_Coil( "axis 1 z" )
   END_RUNG
   RUNG wire#w1
      R_Coil( "Lid alined(1)" )
   END_RUNG
   RUNG wire#w1
      R_Coil( "MOVE Z BIT(1)" )
   END_RUNG
   // the same network as SCL:
   #_w1 := "start memory" AND "IEC_Timer_0_DB_2".Q AND NOT "Tag_10(1)";   // rising edge of "IEC_Timer_0_DB_2".Q
   "Tag_10(1)" := "IEC_Timer_0_DB_2".Q;
   IF #_w1 THEN
       "axis 1 z" := FALSE;
       "Lid alined(1)" := FALSE;
       "MOVE Z BIT(1)" := FALSE;
   END_IF;
END_REGION

REGION Network 5
   RUNG wire#powerrail
      Contact( "start memory" )
      Contact( "axis 1 grab" )
      wire#w1
      N_Contact(operand := "axis 1 z", bit := "Tag_12(1)")
      Contact( "base alined(1)" )
      wire#w2
      S_Coil( "axis 1 x" )
   END_RUNG
   RUNG wire#w1
      I_Contact( "axis 1 moving z" )
   END_RUNG wire#w2
   // the same network as SCL:
   #_w1 := "start memory" AND "axis 1 grab" AND NOT "axis 1 z" AND "Tag_12(1)";   // falling edge of "axis 1 z"
   "Tag_12(1)" := "axis 1 z";
   IF (#_w1 AND "base alined(1)") OR ("start memory" AND "axis 1 grab" AND NOT "axis 1 moving z") THEN
       "axis 1 x" := TRUE;
   END_IF;
END_REGION

REGION Network 6
   RUNG wire#powerrail
      Contact( "start memory" )
      Contact( "axis 1 x" )
      Contact( "axis 1 grab" )
      N_Contact(operand := "axis 1 moving x", bit := "Tag_14(1)")
      wire#w1
      S_Coil( "axis 1 z" )
   END_RUNG
   RUNG wire#w1
      S_Coil( "MOVE Z BIT 2(1)" )
   END_RUNG
   // the same network as SCL:
   #_w1 := "start memory" AND "axis 1 x" AND "axis 1 grab" AND NOT "axis 1 moving x" AND "Tag_14(1)";   // falling edge of "axis 1 moving x"
   "Tag_14(1)" := "axis 1 moving x";
   IF #_w1 THEN
       "axis 1 z" := TRUE;
       "MOVE Z BIT 2(1)" := TRUE;
   END_IF;
END_REGION

REGION Network 7
   RUNG wire#powerrail
      Contact( "start memory" )
      Contact( "axis 1 x" )
      Contact( "axis 1 z" )
      N_Contact(operand := "axis 1 moving z", bit := "Tag_15(1)")
      wire#w1
      R_Coil( "axis 1 grab" )
   END_RUNG
   RUNG wire#w1
      S_Coil( "TEMPORARY(1)" )
   END_RUNG
   RUNG wire#w1
      R_Coil( "base alined(1)" )
   END_RUNG
   // the same network as SCL:
   #_w1 := "start memory" AND "axis 1 x" AND "axis 1 z" AND NOT "axis 1 moving z" AND "Tag_15(1)";   // falling edge of "axis 1 moving z"
   "Tag_15(1)" := "axis 1 moving z";
   IF #_w1 THEN
       "axis 1 grab" := FALSE;
       "TEMPORARY(1)" := TRUE;
       "base alined(1)" := FALSE;
   END_IF;
END_REGION

REGION Network 8
   "IEC_Timer_0_DB_3".TON(IN := "start memory" AND "TEMPORARY(1)", PT := T#1S);
END_REGION

REGION Network 9
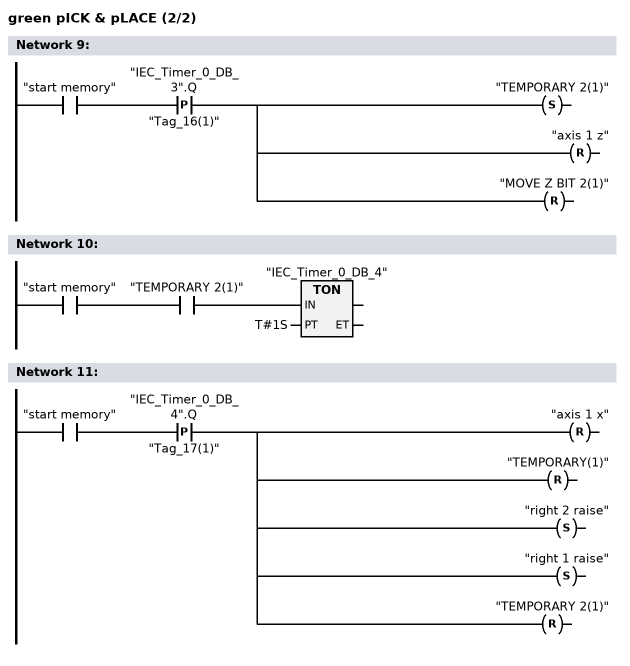
   RUNG wire#powerrail
      Contact( "start memory" )
      P_Contact(operand := "IEC_Timer_0_DB_3".Q, bit := "Tag_16(1)")
      wire#w1
      S_Coil( "TEMPORARY 2(1)" )
   END_RUNG
   RUNG wire#w1
      R_Coil( "axis 1 z" )
   END_RUNG
   RUNG wire#w1
      R_Coil( "MOVE Z BIT 2(1)" )
   END_RUNG
   // the same network as SCL:
   #_w1 := "start memory" AND "IEC_Timer_0_DB_3".Q AND NOT "Tag_16(1)";   // rising edge of "IEC_Timer_0_DB_3".Q
   "Tag_16(1)" := "IEC_Timer_0_DB_3".Q;
   IF #_w1 THEN
       "TEMPORARY 2(1)" := TRUE;
       "axis 1 z" := FALSE;
       "MOVE Z BIT 2(1)" := FALSE;
   END_IF;
END_REGION

REGION Network 10
   "IEC_Timer_0_DB_4".TON(IN := "start memory" AND "TEMPORARY 2(1)", PT := T#1S);
END_REGION

REGION Network 11
   RUNG wire#powerrail
      Contact( "start memory" )
      P_Contact(operand := "IEC_Timer_0_DB_4".Q, bit := "Tag_17(1)")
      wire#w1
      R_Coil( "axis 1 x" )
   END_RUNG
   RUNG wire#w1
      R_Coil( "TEMPORARY(1)" )
   END_RUNG
   RUNG wire#w1
      S_Coil( "right 2 raise" )
   END_RUNG
   RUNG wire#w1
      S_Coil( "right 1 raise" )
   END_RUNG
   RUNG wire#w1
      R_Coil( "TEMPORARY 2(1)" )
   END_RUNG
   // the same network as SCL:
   #_w1 := "start memory" AND "IEC_Timer_0_DB_4".Q AND NOT "Tag_17(1)";   // rising edge of "IEC_Timer_0_DB_4".Q
   "Tag_17(1)" := "IEC_Timer_0_DB_4".Q;
   IF #_w1 THEN
       "axis 1 x" := FALSE;
       "TEMPORARY(1)" := FALSE;
       "right 2 raise" := TRUE;
       "right 1 raise" := TRUE;
       "TEMPORARY 2(1)" := FALSE;
   END_IF;
END_REGION
END_FUNCTION

FUNCTION "MHJ-PLC-Lab-Function-S71500" : Void   // FC9000, SCL
{ S7_Optimized_Access := 'TRUE' }
VERSION : 0.1
   VAR_TEMP
      Value : Byte;
      ForCounter : Int;
   END_VAR
   VAR CONSTANT
      Value_01_DW : DWord := 16#1223_5486;
      Value_02_DW : DWord := 16#A6C9_D1F5;
   END_VAR
BEGIN

   #Value:=PEEK(area := 16#82,
        dbNumber := 0,
        byteOffset := 511);
   #Value := #Value + 1;

   POKE(area := 16#82,
        dbNumber := 0,
        byteOffset := 511,
        value := #Value);

   POKE(area := 16#82,
        dbNumber := 0,
        byteOffset := 1016,
        value := #Value_01_DW);
   POKE(area := 16#82,
        dbNumber := 0,
        byteOffset := 1020,
        value := #Value_02_DW);

   FOR #ForCounter := 0 TO 63 DO
       #Value:=PEEK(area := 16#1,
            dbNumber := 0,
            byteOffset := #ForCounter);
       POKE(area := 16#81,
            dbNumber := 0,
            byteOffset := #ForCounter,
            value := #Value);
   END_FOR;
   #Value := PEEK(area := 16#1,
                  dbNumber := 0,
                  byteOffset := 512);
   POKE(area := 16#82,
        dbNumber := 0,
        byteOffset := 512,
        value := #Value);
END_FUNCTION

ORGANIZATION_BLOCK "Main"   // OB1, LAD, ProgramCycle
TITLE = "Main Program Sweep (Cycle)"
{ S7_Optimized_Access := 'FALSE' }
VERSION : 0.1
   VAR_TEMP
      OB1_EV_CLASS : Byte;   // Bits 0-3 = 1 (Coming event), Bits 4-7 = 1 (Event class 1)
      OB1_SCAN_1 : Byte;   // 1 (Cold restart scan 1 of OB 1), 3 (Scan 2-n of OB 1)
      OB1_PRIORITY : Byte;   // Priority of OB Execution
      OB1_OB_NUMBR : Byte;   // 1 (Organization block 1, OB1)
      OB1_RESERVED_1 : Byte;   // Reserved for system
      OB1_RESERVED_2 : Byte;   // Reserved for system
      OB1_PREV_CYCLE : Int;   // Cycle time of previous OB1 scan (milliseconds)
      OB1_MIN_CYCLE : Int;   // Minimum cycle time of OB1 (milliseconds)
      OB1_MAX_CYCLE : Int;   // Maximum cycle time of OB1 (milliseconds)
      OB1_DATE_TIME : Date_And_Time;   // Date and time OB1 started
   END_VAR
   VAR_TEMP   // added for the SCL form of the ladder/FBD networks
      _w1 : Bool;
   END_VAR
BEGIN

REGION Network 1: connection Function block
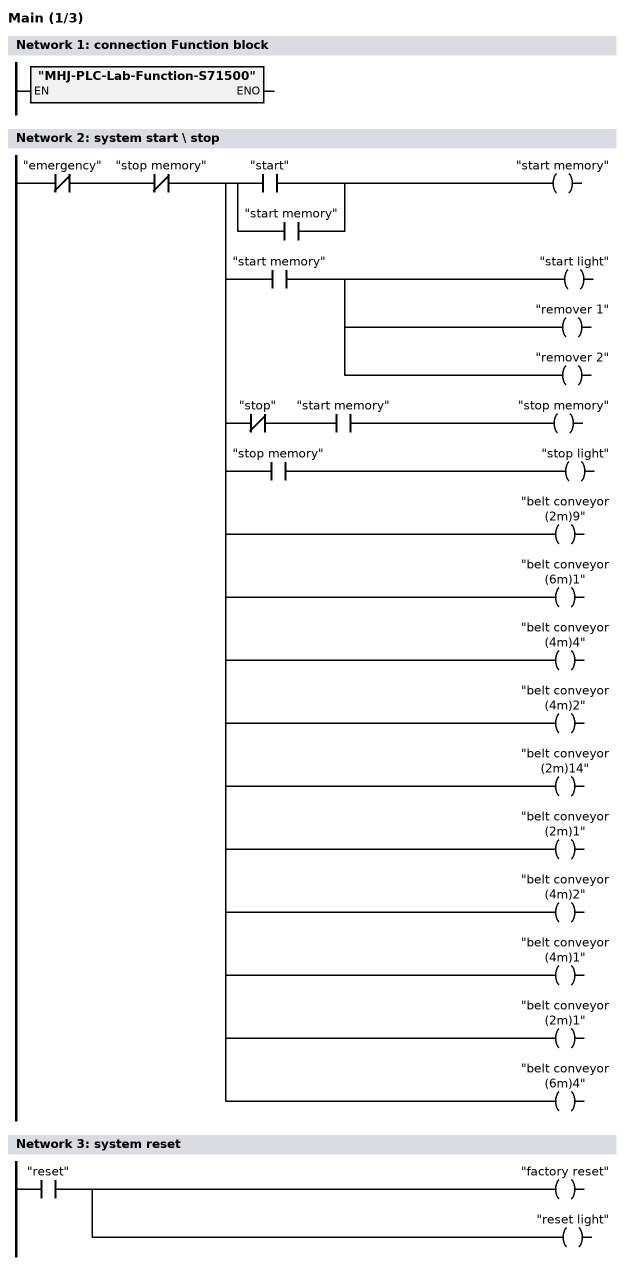
   RUNG wire#powerrail
      "MHJ-PLC-Lab-Function-S71500"()
   END_RUNG
   // the same network as SCL:
   "MHJ-PLC-Lab-Function-S71500"();
END_REGION

REGION Network 2: system start \ stop
   RUNG wire#powerrail
      I_Contact( "emergency" )
      I_Contact( "stop memory" )
      wire#w1
      Contact( "start" )
      wire#w2
      Coil( "start memory" )
   END_RUNG
   RUNG wire#w1
      Contact( "start memory" )
   END_RUNG wire#w2
   RUNG wire#w1
      Contact( "start memory" )
      wire#w3
      Coil( "start light" )
   END_RUNG
   RUNG wire#w3
      Coil( "remover 1" )
   END_RUNG
   RUNG wire#w3
      Coil( "remover 2" )
   END_RUNG
   RUNG wire#w1
      I_Contact( "stop" )
      Contact( "start memory" )
      Coil( "stop memory" )
   END_RUNG
   RUNG wire#w1
      Contact( "stop memory" )
      Coil( "stop light" )
   END_RUNG
   RUNG wire#w1
      Coil( "belt conveyor (2m)9" )
   END_RUNG
   RUNG wire#w1
      Coil( "belt conveyor (6m)1" )
   END_RUNG
   RUNG wire#w1
      Coil( "belt conveyor (4m)4" )
   END_RUNG
   RUNG wire#w1
      Coil( "belt conveyor (4m)2" )
   END_RUNG
   RUNG wire#w1
      Coil( "belt conveyor (2m)14" )
   END_RUNG
   RUNG wire#w1
      Coil( "belt conveyor (2m)1" )
   END_RUNG
   RUNG wire#w1
      Coil( "belt conveyor (4m)2" )
   END_RUNG
   RUNG wire#w1
      Coil( "belt conveyor (4m)1" )
   END_RUNG
   RUNG wire#w1
      Coil( "belt conveyor (2m)1" )
   END_RUNG
   RUNG wire#w1
      Coil( "belt conveyor (6m)4" )
   END_RUNG
   // the same network as SCL:
   #_w1 := NOT "emergency" AND NOT "stop memory";
   "start memory" := #_w1 AND ("start" OR "start memory");
   "start light" := #_w1 AND "start memory";
   "remover 1" := "start light";
   "remover 2" := "start light";
   "stop memory" := #_w1 AND NOT "stop" AND "start memory";
   "stop light" := #_w1 AND "stop memory";
   "belt conveyor (2m)9" := #_w1;
   "belt conveyor (6m)1" := #_w1;
   "belt conveyor (4m)4" := #_w1;
   "belt conveyor (4m)2" := #_w1;
   "belt conveyor (2m)14" := #_w1;
   "belt conveyor (2m)1" := #_w1;
   "belt conveyor (4m)2" := #_w1;
   "belt conveyor (4m)1" := #_w1;
   "belt conveyor (2m)1" := #_w1;
   "belt conveyor (6m)4" := #_w1;
END_REGION

REGION Network 3: system reset
   RUNG wire#powerrail
      Contact( "reset" )
      wire#w1
      Coil( "factory reset" )
   END_RUNG
   RUNG wire#w1
      Coil( "reset light" )
   END_RUNG
   // the same network as SCL:
   "factory reset" := "reset";
   "reset light" := "reset";
END_REGION

REGION Network 4: reset machining station
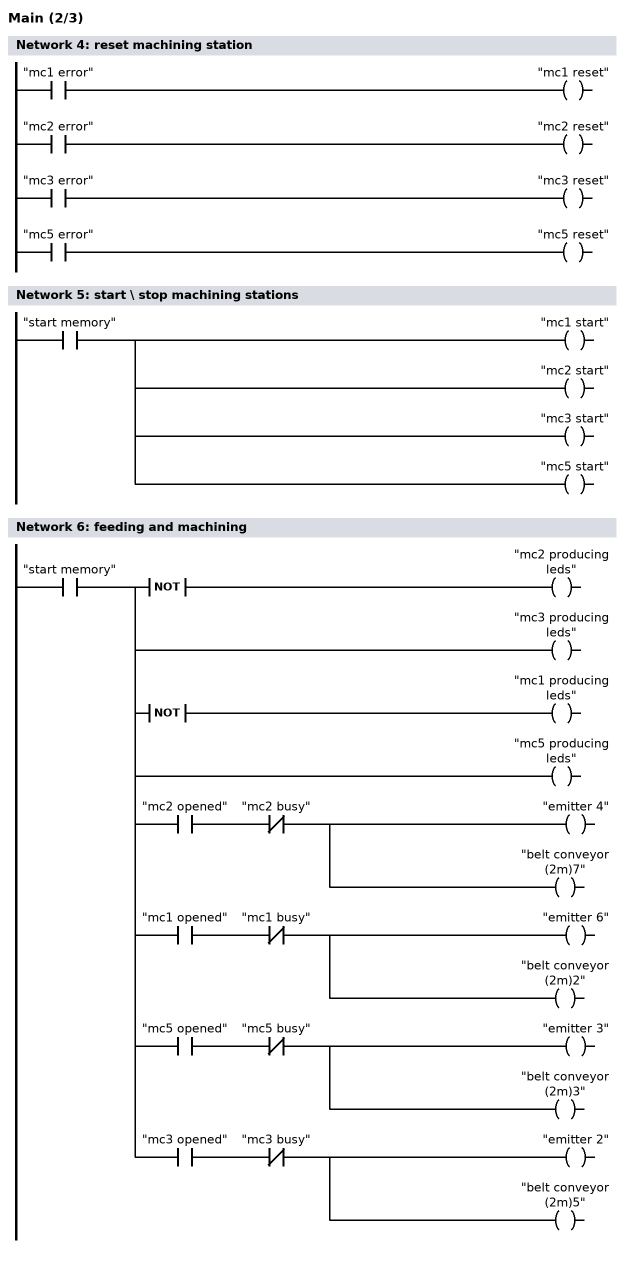
   RUNG wire#powerrail
      Contact( "mc1 error" )
      Coil( "mc1 reset" )
   END_RUNG
   RUNG wire#powerrail
      Contact( "mc2 error" )
      Coil( "mc2 reset" )
   END_RUNG
   RUNG wire#powerrail
      Contact( "mc3 error" )
      Coil( "mc3 reset" )
   END_RUNG
   RUNG wire#powerrail
      Contact( "mc5 error" )
      Coil( "mc5 reset" )
   END_RUNG
   // the same network as SCL:
   "mc1 reset" := "mc1 error";
   "mc2 reset" := "mc2 error";
   "mc3 reset" := "mc3 error";
   "mc5 reset" := "mc5 error";
END_REGION

REGION Network 5: start \ stop machining stations
   RUNG wire#powerrail
      Contact( "start memory" )
      wire#w1
      Coil( "mc1 start" )
   END_RUNG
   RUNG wire#w1
      Coil( "mc2 start" )
   END_RUNG
   RUNG wire#w1
      Coil( "mc3 start" )
   END_RUNG
   RUNG wire#w1
      Coil( "mc5 start" )
   END_RUNG
   // the same network as SCL:
   "mc1 start" := "start memory";
   "mc2 start" := "start memory";
   "mc3 start" := "start memory";
   "mc5 start" := "start memory";
END_REGION

REGION Network 6: feeding and machining
   RUNG wire#powerrail
      Contact( "start memory" )
      wire#w1
      Not()
      Coil( "mc2 producing leds" )
   END_RUNG
   RUNG wire#w1
      Coil( "mc3 producing leds" )
   END_RUNG
   RUNG wire#w1
      Not()
      Coil( "mc1 producing leds" )
   END_RUNG
   RUNG wire#w1
      Coil( "mc5 producing leds" )
   END_RUNG
   RUNG wire#w1
      Contact( "mc2 opened" )
      I_Contact( "mc2 busy" )
      wire#w2
      Coil( "emitter 4" )
   END_RUNG
   RUNG wire#w2
      Coil( "belt conveyor (2m)7" )
   END_RUNG
   RUNG wire#w1
      Contact( "mc1 opened" )
      I_Contact( "mc1 busy" )
      wire#w3
      Coil( "emitter 6" )
   END_RUNG
   RUNG wire#w3
      Coil( "belt conveyor (2m)2" )
   END_RUNG
   RUNG wire#w1
      Contact( "mc5 opened" )
      I_Contact( "mc5 busy" )
      wire#w4
      Coil( "emitter 3" )
   END_RUNG
   RUNG wire#w4
      Coil( "belt conveyor (2m)3" )
   END_RUNG
   RUNG wire#w1
      Contact( "mc3 opened" )
      I_Contact( "mc3 busy" )
      wire#w5
      Coil( "emitter 2" )
   END_RUNG
   RUNG wire#w5
      Coil( "belt conveyor (2m)5" )
   END_RUNG
   // the same network as SCL:
   "mc2 producing leds" := NOT "start memory";
   "mc3 producing leds" := "start memory";
   "mc1 producing leds" := NOT "start memory";
   "mc5 producing leds" := "start memory";
   "emitter 4" := "start memory" AND "mc2 opened" AND NOT "mc2 busy";
   "belt conveyor (2m)7" := "emitter 4";
   "emitter 6" := "start memory" AND "mc1 opened" AND NOT "mc1 busy";
   "belt conveyor (2m)2" := "emitter 6";
   "emitter 3" := "start memory" AND "mc5 opened" AND NOT "mc5 busy";
   "belt conveyor (2m)3" := "emitter 3";
   "emitter 2" := "start memory" AND "mc3 opened" AND NOT "mc3 busy";
   "belt conveyor (2m)5" := "emitter 2";
END_REGION

REGION Network 7: Sorting
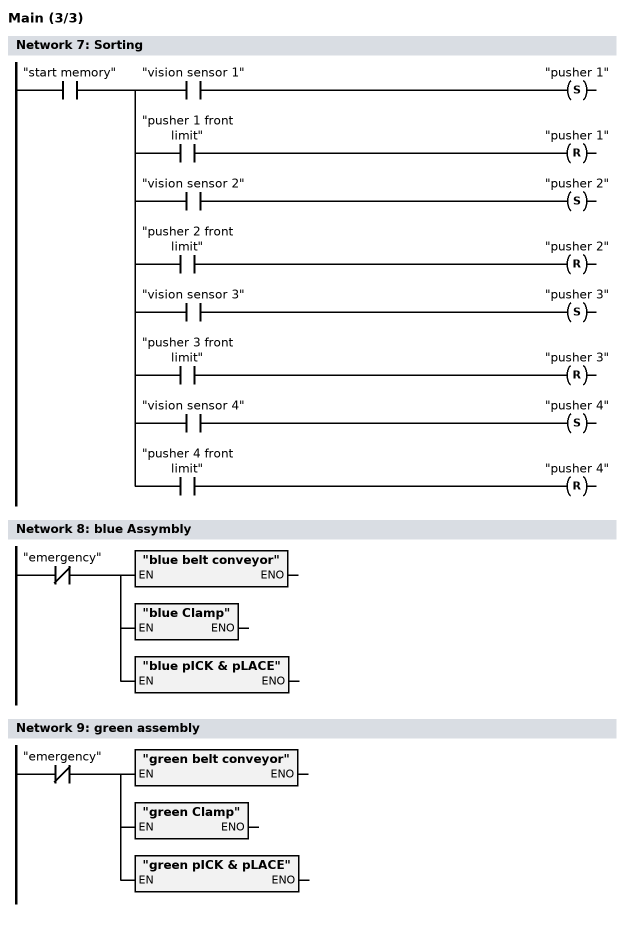
   RUNG wire#powerrail
      Contact( "start memory" )
      wire#w1
      Contact( "vision sensor 1" )
      S_Coil( "pusher 1" )
   END_RUNG
   RUNG wire#w1
      Contact( "pusher 1 front limit" )
      R_Coil( "pusher 1" )
   END_RUNG
   RUNG wire#w1
      Contact( "vision sensor 2" )
      S_Coil( "pusher 2" )
   END_RUNG
   RUNG wire#w1
      Contact( "pusher 2 front limit" )
      R_Coil( "pusher 2" )
   END_RUNG
   RUNG wire#w1
      Contact( "vision sensor 3" )
      S_Coil( "pusher 3" )
   END_RUNG
   RUNG wire#w1
      Contact( "pusher 3 front limit" )
      R_Coil( "pusher 3" )
   END_RUNG
   RUNG wire#w1
      Contact( "vision sensor 4" )
      S_Coil( "pusher 4" )
   END_RUNG
   RUNG wire#w1
      Contact( "pusher 4 front limit" )
      R_Coil( "pusher 4" )
   END_RUNG
   // the same network as SCL:
   IF "start memory" AND "vision sensor 1" THEN "pusher 1" := TRUE; END_IF;
   IF "start memory" AND "pusher 1 front limit" THEN "pusher 1" := FALSE; END_IF;
   IF "start memory" AND "vision sensor 2" THEN "pusher 2" := TRUE; END_IF;
   IF "start memory" AND "pusher 2 front limit" THEN "pusher 2" := FALSE; END_IF;
   IF "start memory" AND "vision sensor 3" THEN "pusher 3" := TRUE; END_IF;
   IF "start memory" AND "pusher 3 front limit" THEN "pusher 3" := FALSE; END_IF;
   IF "start memory" AND "vision sensor 4" THEN "pusher 4" := TRUE; END_IF;
   IF "start memory" AND "pusher 4 front limit" THEN "pusher 4" := FALSE; END_IF;
END_REGION

REGION Network 8: blue Assymbly
   RUNG wire#powerrail
      I_Contact( "emergency" )
      wire#w1
      "blue belt conveyor"()
   END_RUNG
   RUNG wire#w1
      "blue Clamp"()
   END_RUNG
   RUNG wire#w1
      "blue pICK & pLACE"()
   END_RUNG
   // the same network as SCL:
   #_w1 := NOT "emergency";
   IF #_w1 THEN
       "blue belt conveyor"();
       "blue Clamp"();
       "blue pICK & pLACE"();
   END_IF;
END_REGION

REGION Network 9: green assembly
   RUNG wire#powerrail
      I_Contact( "emergency" )
      wire#w1
      "green belt conveyor"()
   END_RUNG
   RUNG wire#w1
      "green Clamp"()
   END_RUNG
   RUNG wire#w1
      "green pICK & pLACE"()
   END_RUNG
   // the same network as SCL:
   #_w1 := NOT "emergency";
   IF #_w1 THEN
       "green belt conveyor"();
       "green Clamp"();
       "green pICK & pLACE"();
   END_IF;
END_REGION
END_ORGANIZATION_BLOCK